PROGRAM MAIN
VAR
	axisRef				: AXIS_REF;
	fbAxisControl		: MC_AxisControl;
END_VAR

fbAxisControl(axisRef:= axisRef);

END_PROGRAM

(* stored: Version 1.1.0.1, ProductVersion 3.1.4024.9
   POU MAIN: Id {7f1c0017-b14e-4b9f-8e23-d981db59398c}, SpecialFunc None *)
